RoboDK station: drilling.rdk

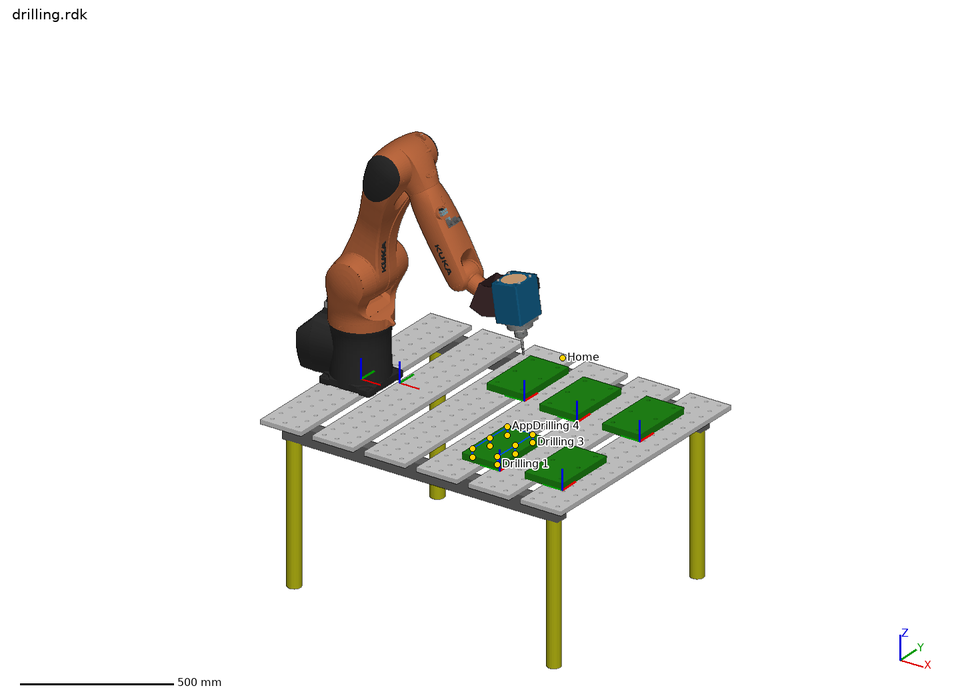
[picture v0: the station drawn from its stored meshes, robots at their saved joint values, targets as dots, program paths as lines]
Station Drilling (saved by RoboDK 5.8.0). Poses are relative to the parent item; angles as X-Y-Z fixed-axis rotations.
  - frame KUKA KR 10 R900 sixx Base at (-120, 10, 0) mm
    - robot KUKA KR 10 R900 sixx: 6 axes, payload 10 kg, reach 901 mm, repeatability 0.03 mm, weight 52 kg
        modified DH rows (alpha deg, a mm, theta deg, d mm): 0, 0, 0, 400; -90, 25, 0, 0; 0, 455, -90, 0; -90, 35, 0, 420; 90, 0, 0, 0; -90, 0, 180, 80
        joint limits [-170, -190, -120, -185, -120, -350] to [170, 45, 156, 185, 120, 350]; home [0, -90, 90, 0, 0, 0]; saved at [0, -71.953, 131.164, 0, -37.509, 0]
      - tool Spindle, TCP at (116.06, 0, 219.48) mm, rotated rx 0 ry 60 rz 0 deg, size 260.9 x 152 x 222 mm, geometry from Little spindle.step
  - frame Frame World at (0, 60, 0) mm
    - target Home (Cartesian target) at (646.35, 0, 271.16) mm, rotated rx 180 ry 8.3 rz -180 deg; joints [0, -72.5, 126.226, 0, -25.229, 0] of KUKA KR 10 R900 sixx
    - object Table at (380, 0, 0) mm, size 1193.8 x 965.2 x 609.6 mm, geometry from welding_table.sld
  - frame Part 1 at (640.29, -290, 0) mm, rotated rx 0 ry 0 rz 90 deg
    - object Drilling Part 1 at (0, 0, 0) mm, size 250 x 150 x 25 mm, geometry from Drilling.step
      - object Drilling Part 1 at (0, 0, 0) mm, size 250 x 150 x 25 mm, geometry from Drilling.step
    - target Drilling 1 (Cartesian target) at (25, 25, 5) mm, rotated rx -180 ry 0 rz 90 deg; joints [9.438, -40.7, 124.04, 9.501, -83.43, -1.097] of KUKA KR 10 R900 sixx
    - target Drilling 2 (Cartesian target) at (125, 25, 5) mm, rotated rx -180 ry 0 rz 90 deg; joints [-57.379, -35.838, 153.204, -126.861, -32.652, -27.341] of KUKA KR 10 R900 sixx
    - target Drilling 3 (Cartesian target) at (225, 25, 5) mm, rotated rx -180 ry 0 rz 90 deg; joints [-40.958, -39.896, 145.068, -120.051, -44.318, -16.433] of KUKA KR 10 R900 sixx
    - target Drilling 4 (Cartesian target) at (225, 125, 5) mm, rotated rx -180 ry 0 rz 90 deg; joints [-52.695, -41.042, 135.387, -140.548, -49.797, -3.447] of KUKA KR 10 R900 sixx
    - target Drilling 5 (Cartesian target) at (125, 125, 5) mm, rotated rx -180 ry 0 rz 90 deg; joints [-67.057, -40.548, 142.134, -152.596, -42.703, -6.629] of KUKA KR 10 R900 sixx
    - target Drilling 6 (Cartesian target) at (25, 125, 5) mm, rotated rx -180 ry 0 rz 90 deg; joints [-85.161, -39.839, 145.27, 6.321, 37.844, 177.903] of KUKA KR 10 R900 sixx
    - target AppDrilling 1 (Cartesian target) at (25, 25, 35) mm, rotated rx -180 ry 0 rz 90 deg; joints [9.438, -44.943, 125.087, 9.577, -80.279, -1.632] of KUKA KR 10 R900 sixx
    - target AppDrilling 2 (Cartesian target) at (125, 25, 35) mm, rotated rx -180 ry 0 rz 90 deg; joints [-57.379, -42.811, 155.1, -132.596, -35.902, -20.405] of KUKA KR 10 R900 sixx
    - target AppDrilling 3 (Cartesian target) at (225, 25, 35) mm, rotated rx -180 ry 0 rz 90 deg; joints [-40.958, -45.85, 146.604, -123.74, -46.654, -11.173] of KUKA KR 10 R900 sixx
    - target AppDrilling 4 (Cartesian target) at (225, 125, 35) mm, rotated rx -180 ry 0 rz 90 deg; joints [-52.695, -46.066, 136.671, -142.417, -52.723, -0.461] of KUKA KR 10 R900 sixx
    - target AppDrilling 5 (Cartesian target) at (125, 125, 35) mm, rotated rx -180 ry 0 rz 90 deg; joints [-67.057, -46.187, 143.58, -154.493, -46.459, -3.968] of KUKA KR 10 R900 sixx
    - target AppDrilling 6 (Cartesian target) at (25, 125, 35) mm, rotated rx -180 ry 0 rz 90 deg; joints [-85.161, -45.815, 146.813, 5.766, 42.253, 178.629] of KUKA KR 10 R900 sixx
  - frame Part 2 at (640.29, 150, 0) mm, rotated rx 0 ry 0 rz 90 deg
    - object Drilling Part 2 at (0, 0, 0) mm, size 250 x 150 x 25 mm, geometry from Drilling.step
  - frame Part 3 at (890.29, 150, 0) mm, rotated rx 0 ry 0 rz 90 deg
    - object Drilling Part 3 at (0, 0, 0) mm, size 250 x 150 x 25 mm, geometry from Drilling.step
  - frame Part 4 at (890.29, -290, 0) mm, rotated rx 0 ry 0 rz 90 deg
    - object Drilling Part 4 at (0, 0, 0) mm, size 250 x 150 x 25 mm, geometry from Drilling.step
  - frame Part 5 at (410.29, 180, 0) mm, rotated rx 0 ry 0 rz 90 deg
    - object Drilling Part 5 at (0, 0, 0) mm, size 250 x 150 x 25 mm, geometry from Drilling.step
  - program Test (7 instructions, listed below)
  - program DrillProgram1 (2 instructions, listed below)
  - program DrillProgram2 (2 instructions, listed below)
  - program DrillProgram3 (3 instructions, listed below)
  - program DrillProgram4 (2 instructions, listed below)
  - program DrillProgram5 (2 instructions, listed below)
  - program GoHome (3 instructions, listed below)
  - program DrillingPart (19 instructions, listed below)
  - Python program RunProgram (listed below)
  - program Main (6 instructions, listed below)
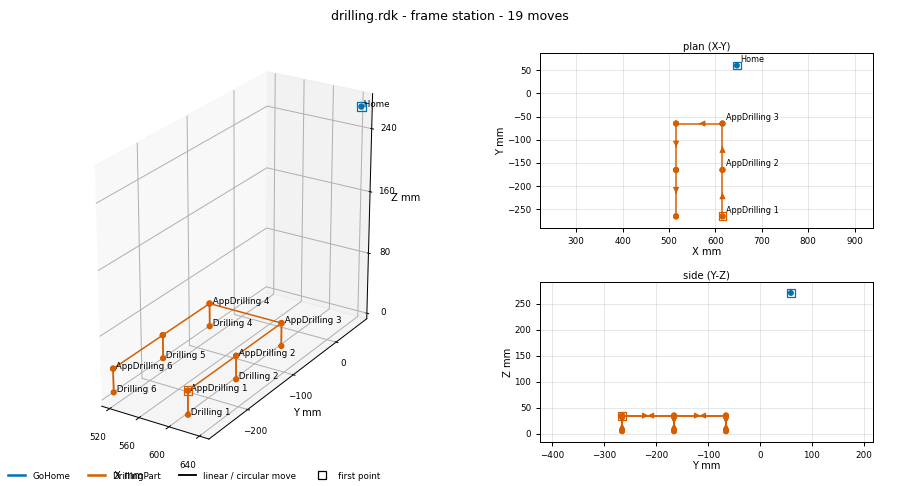
[picture p0: tool path of drilling.rdk in frame station, 19 of 19 moves have a stored position in this frame; points joined in program order, loops and branches not executed]

--- program Test (robot KUKA KR 10 R900 sixx) ---
  Call GoHome
  Set Ref.: Part 1
  Call DrillingPart
  Call GoHome
  Call DrillingPart
  Set Ref.: Part 2
  Call GoHome

--- program DrillProgram1 (robot KUKA KR 10 R900 sixx) ---
  Set Ref.: Part 1
  Call DrillingPart

--- program DrillProgram2 (robot KUKA KR 10 R900 sixx) ---
  Set Ref.: Part 2
  Call DrillingPart

--- program DrillProgram3 (robot KUKA KR 10 R900 sixx) ---
  Call GoHome
  Set Ref.: Part 3
  Call DrillingPart

--- program DrillProgram4 (robot KUKA KR 10 R900 sixx) ---
  Set Ref.: Part 4
  Call DrillingPart

--- program DrillProgram5 (robot KUKA KR 10 R900 sixx) ---
  Set Ref.: Part 5
  Call DrillingPart

--- program GoHome (robot KUKA KR 10 R900 sixx) ---
  Set Ref.: KUKA KR 10 R900 sixx Base
  Set Tool: Spindle
  MoveJ (Home)

--- program DrillingPart (robot KUKA KR 10 R900 sixx) ---
  Set Tool: Spindle
  MoveL (AppDrilling 1)
  MoveL (Drilling 1)
  MoveL (AppDrilling 1)
  MoveL (AppDrilling 2)
  MoveL (Drilling 2)
  MoveL (AppDrilling 2)
  MoveL (AppDrilling 3)
  MoveL (Drilling 3)
  MoveL (AppDrilling 3)
  MoveL (AppDrilling 4)
  MoveL (Drilling 4)
  MoveL (AppDrilling 4)
  MoveL (AppDrilling 5)
  MoveL (Drilling 5)
  MoveL (AppDrilling 5)
  MoveL (AppDrilling 6)
  MoveL (Drilling 6)
  MoveL (AppDrilling 6)

--- Python program RunProgram ---
# This macro shows how to run a program as an event (right click an object and select Run Program)
# Events must be listed in Edit Events menu from the object menu
# (double click an object, select More Options and Edit Events)
# You can list the events as Name -> Script
from robolink import *    # API to communicate with RoboDK
from robodk import *      # basic matrix operations
RDK = Robolink()

item = None

# Check if we are running this program inside another program and passing arguments
import sys
if len(sys.argv) > 1:
    item_name = sys.argv[1]
    item = RDK.Item(item_name)

# If the default ACTION is None, display a message to activate/deactivate the spray gun
if item is None or not item.Valid():
    print('Note: This macro can be called as RunProgram("Drilling Part 1")')
    item = RDK.ItemUserPick("Select an object", ITEM_TYPE_OBJECT)

if item is None or not item.Valid():
    print("User selected cancel or an invalid program")
    quit()

item_name = item.Name()

# The object name will be Drilling Part 1 or Drilling Part 2
# Get the last ID to call the corresponding program DrillProgram1 or DrillProgram2
name_words = item_name.split(' ')

try:
    prog_id = int(name_words[-1])
    program_name = "DrillProgram" + str(prog_id)

except ValueError:
    # Use MainProgram if we select the table or an object without a number
    program_name = "MainProgram"

# Retrieve the program by name
program = RDK.Item(program_name, ITEM_TYPE_PROGRAM)

if not program.Valid():
    RDK.ShowMessage("Program not found: " + program_name)
    quit()

program.RunProgram()

--- program Main (robot KUKA KR 10 R900 sixx) ---
  Call DrillProgram3
  Call DrillProgram4
  Call DrillProgram1
  Call DrillProgram2
  Call DrillProgram5
  Call GoHome
